Fanuc KAREL source: kb00052.KL

PROGRAM KB00052
%STACKSIZE=65535
%PRIORITY=65535
%NOLOCKGROUP
VAR
P1 : INTEGER
P2 : INTEGER
RESULT : XYZWPREXT
BEGIN
P1=1
P2=1
-- UNRESOLVED_PC line 10 opcodes [27 22 22 27 9D 76 7E 4A] marker_code=24
END KB00052
